Fanuc KAREL source: kb00108.KL

-- PROVISIONAL review KL for V1013-1; original PC SHA256 75a0f1fa51e949b02acff816e39d7bc37bb0f2d39709720c19de9daa078bbedc
-- Incomplete behavior may be omitted. Consult companion uncertainty JSON. Do not deploy.
PROGRAM KB00108
%NOLOCKGROUP
BEGIN
  -- UNRESOLVED_PC offsets 5-12; opcodes 9D,23
  -- UNRESOLVED_PC offsets 17-24; opcodes 9D,23
  -- UNRESOLVED_PC offsets 29-39; opcodes 9D,22,9D,33,35
  -- UNRESOLVED_PC offsets 44-51; opcodes 9D,23
  -- UNRESOLVED_PC offsets 56-90; opcodes 27,22,22,22,22,22,31
  -- UNRESOLVED_PC offsets 95-99; opcodes 7F
END KB00108
